SUBAPPLICATION AR_M2M_Subscribe_TO_Q_Publish_OPC (* Remote-Subscribe eines bereits fertigen physikalischen Werts (M2M, von einer anderen Station) -> VT-Anzeige (Q_NumericValue_PHYSA) UND lokaler Re-Publish (fuer weitere lokale Konsumenten/Web-Mirror/Dashboard). Ersetzt AR_HZ_TO_Q_Publish_OPC fuer Sensoren, deren Hz->Einheit-Umrechnung jetzt lokal auf der Sensor-Station laeuft (logiBUS_PI_Speed_Publish_OPC) statt hier zentral - kein SCALE/AR_MUL_2 mehr noetig, nur noch Subscribe+Anzeige+Re-Publish. *)
  (* Standard: 61499-2; Description: Copyright (c) 2026 Meisterschulen am Ostbahnhof This program and the accompanying materials are made available under the terms of the Eclipse Public License 2.0 which is available at https://www.eclipse.org/legal/epl-2.0/ SPDX-License-Identifier: EPL-2.0 *)
  (* Version 1.0, 2026-09-17, Franz Höpfinger, Meisterschulen am Ostbahnhof, initial implementation - schlanke Nachfolge-Variante von AR_HZ_TO_Q_Publish_OPC ohne eigene Skalierung, da die Hz->Einheit-Umrechnung jetzt auf der Sensor-Station selbst laeuft (logiBUS_PI_Speed_Publish_OPC). Buendelt AR_SUBSCRIBE_1+AR_TO_Q_Publish_OPC - ein Baustein je bereits umgerechnetem Puls-/Analog-Wert, der von einer anderen Station remote abonniert wird. *)
  (* Version 1.1, 2026-09-21, Franz Höpfinger, Meisterschulen am Ostbahnhof, Neuer Plug VALUE_OUT (AR) ergaenzt - Fuellband-Winkel-Migration (Kalibrierung zieht auf die Sensor-Station um) braucht den remote abonnierten Wert nicht nur fuer die VT-Anzeige/den eigenen Re-Publish, sondern auch als direkten AR-Plug fuer weitere lokale Konsumenten (Befuellautomatik/Fuellband_Oben) - analog zum bereits etablierten VALUE_OUT-Muster in NumericValue_TO_AR2_OPC v1.1. AR_SPLIT_2 vor Publish.AR_IN eingefuegt, statt AR_SUBSCRIBE_M2M.OUT direkt dorthin zu verdrahten. *)
  PACKAGE MyLib::sys;
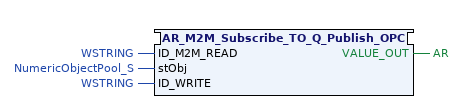
  VAR_INPUT
    ID_M2M_READ : WSTRING; (* Remote-Subscribe-Adresse des bereits fertigen physikalischen Werts (REAL), z.B. FBs::Ventilsteuerung::Ventilsteuerung_STG1::RemoteSubStrings::AUFNAHME_GESCHWINDIGKEIT_KMH_M2M *)
    stObj : logiBUS::utils::conversion::phys::NumericObjectPool_S; (* Object pool properties der VT-Zahlenvariable (u16ObjId, scale, offset, decimals) - z.B. FBs::const::DefaultPool_Numeric::NumberVariable_X_N *)
    ID_WRITE : WSTRING; (* Lokale Publish-Adresse (REAL, physikalischer Wert) - Web-Mirror/Dashboard/Self-Subscribe weiterer lokaler Konsumenten *)
  END_VAR
  PLUGS
    VALUE_OUT : adapter::types::unidirectional::AR; (* Nur-Lese-Spiegel des remote abonnierten Werts, fuer weitere lokale Konsumenten (SubApp-Sockets statt eigenem OPC-UA-Self-Subscribe) - vermeidet Doppel-Self-Subscribe desselben Remote-Knotens auf dieser Station *)
  END_PLUGS
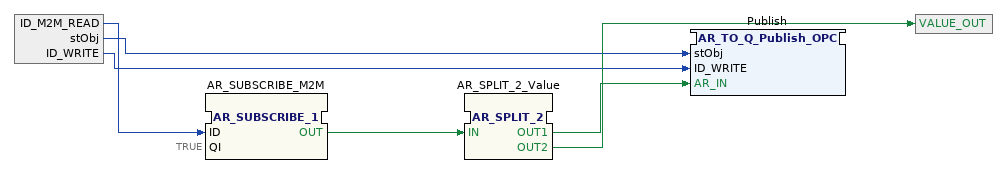
  FBS
    AR_SUBSCRIBE_M2M : adapter::net::AR_SUBSCRIBE_1(QI := TRUE);
    AR_SPLIT_2_Value : adapter::events::unidirectional::AR_SPLIT_2;
  END_FBS
  SUBAPPS
    Publish : MyLib::sys::AR_TO_Q_Publish_OPC;
  END_SUBAPPS
  DATA_CONNECTIONS
    ID_M2M_READ TO AR_SUBSCRIBE_M2M.ID;
    stObj TO Publish.stObj;
    ID_WRITE TO Publish.ID_WRITE;
  END_CONNECTIONS
  ADAPTER_CONNECTIONS
    AR_SUBSCRIBE_M2M.OUT TO AR_SPLIT_2_Value.IN;
    AR_SPLIT_2_Value.OUT1 TO Publish.AR_IN;
    AR_SPLIT_2_Value.OUT2 TO VALUE_OUT;
  END_CONNECTIONS
END_SUBAPPLICATION
